FUNCTION_BLOCK FB_Rectangle IMPLEMENTS I_Shape
VAR_INPUT
END_VAR
VAR_OUTPUT
END_VAR
VAR
	rLength : REAL;
	rWidth : REAL;
END_VAR

METHOD CalculateArea : REAL
VAR_INPUT
END_VAR
CalculateArea := rLength * rWidth;
END_METHOD

PROPERTY Length : REAL
GET
Length := rLength;
END_GET
SET
rLength := Length;
END_SET
END_PROPERTY

PROPERTY Width : REAL
GET
Width := rWidth;
END_GET
SET
rWidth := Width;
END_SET
END_PROPERTY

END_FUNCTION_BLOCK

(* stored: Version 1.1.0.1, ProductVersion 3.1.4024.13
   POU FB_Rectangle: Id {14c618ee-54da-4b99-9f7b-017562a1a7a2}, SpecialFunc None
   Method CalculateArea: Id {8dd0b452-85fb-4a49-b1f2-c11d2d6b033d}
   Property Length: Id {7dc5cff2-e264-45ff-aef8-8525cc5d278e}
   Get Get: Id {4303b057-28a7-4406-9c53-d07215875fbd}
   Set Set: Id {97db6bbb-659f-409a-9ca9-4a4e3956d1f5}
   Property Width: Id {b6576844-1967-4394-8bd5-183c8dbcdfcc}
   Get Get: Id {f8b31081-aae4-47db-b342-662716b20329}
   Set Set: Id {7db4cb98-da03-4beb-92bd-1ed6ce5abb1b} *)
